Fanuc KAREL source: port_FLG.kl

PROGRAM TP
%NOLOCKGROUP
VAR
 x: BOOLEAN
BEGIN
 x = FLG[3]
END TP
